{attribute 'GeneratedUsingTerminal: EL1008-0000-0018'}
{attribute addProperty VendorId "#x00000002"}
{attribute addProperty BoxType "EL1008-0000-0018"}
{attribute addProperty Description "EL1008 8Ch. Dig. Input 24V, 3ms"}
{attribute addProperty Physics "KK"}
{attribute addProperty Id "Channel_1AT %I*Channel_830843C11Channel_2AT %I*Channel_830843C11Channel_3AT %I*Channel_830843C11Channel_4AT %I*Channel_830843C11Channel_5AT %I*Channel_830843C11Channel_6AT %I*Channel_830843C11Channel_7AT %I*Channel_830843C11Channel_8AT %I*Channel_830843C11WcStateAT %I*WcState_9091E0EB2InfoDataAT %I*InfoData_6F19DB2B2"}
{attribute addProperty CRC "2028524509"}
{attribute addProperty Size "12"}
TYPE EL1008_78E8D3DD EXTENDS TcoIo.EtcSlaveTerminalBase_947E5A46 : STRUCT
    {attribute addProperty Name "Channel_1"}
    Channel_1 : Channel_830843C1;
    {attribute addProperty Name "Channel_2"}
    Channel_2 : Channel_830843C1;
    {attribute addProperty Name "Channel_3"}
    Channel_3 : Channel_830843C1;
    {attribute addProperty Name "Channel_4"}
    Channel_4 : Channel_830843C1;
    {attribute addProperty Name "Channel_5"}
    Channel_5 : Channel_830843C1;
    {attribute addProperty Name "Channel_6"}
    Channel_6 : Channel_830843C1;
    {attribute addProperty Name "Channel_7"}
    Channel_7 : Channel_830843C1;
    {attribute addProperty Name "Channel_8"}
    Channel_8 : Channel_830843C1;
    {attribute addProperty Name "WcState"}
    WcState : TcoIo.WcState_9091E0EB;
    {attribute addProperty Name "InfoData"}
    InfoData : TcoIo.InfoData_6F19DB2B;
END_STRUCT
END_TYPE

(* stored: Version 1.2.0.0, ProductVersion 3.1.4024.12
   DUT EL1008_78E8D3DD: Id {dff4ea31-1acc-0057-1828-6d41cbd31d42} *)
